// TIA Portal V16 export
// export: Created 2021-09-08T12:44:31.902824Z, ExportSetting WithDefaults, DisplayName Totally Integrated Automation Portal, DisplayVersion V16 Update 3, DisplayName TIA Portal Version Control Interface, DisplayVersion V16 Update 2, DisplayName TIA Portal Openness, DisplayVersion V16 Update 3, DisplayName TIA Portal Teamcenter Gateway, DisplayVersion V16, DisplayName STEP 7 Professional, DisplayVersion V16 Update 3, DisplayName STEP 7 Safety, DisplayVersion V16, DisplayName WinCC Advanced, DisplayVersion V16 Update 3
VAR_GLOBAL   // PLC tag table "A1_AI"
   aiDVA503_Pos AT %IW64 : Int;   // DVA503 Завдання
   aiDVA510_Pos AT %IW66 : Int;   // DVA510 Завдання
END_VAR
VAR_GLOBAL CONSTANT   // user constants
   "iwDVA-503_Setting" : Int := 0;
   "iwDVA-510_Setting" : Int := 1;
END_VAR
